TYPE csp_case_closing_rfid_status_enum :
(
	CSP_CASE_CLOSING_RFID_STATUS_START									:= 5,
	CSP_CASE_CLOSING_RFID_STATUS_ENABLED								:= 6,
	CSP_CASE_CLOSING_RFID_STATUS_PADDLES_START							:= 10,
	CSP_CASE_CLOSING_RFID_STATUS_VERIFY_AXIS_SAFE_POS					:= 15,
	CSP_CASE_CLOSING_RFID_STATUS_UPPER_START 							:= 20,
	CSP_CASE_CLOSING_RFID_STATUS_UPPER_VERIFY_AXIS_POS					:= 25,
	CSP_CASE_CLOSING_RFID_STATUS_UPPER_READ_START						:= 30,
	CSP_CASE_CLOSING_RFID_STATUS_UPPER_READ_CHECK_RESULT				:= 35,
	CSP_CASE_CLOSING_RFID_STATUS_UPPER_RETURN_TO_SAFE_POS				:= 40,
	CSP_CASE_CLOSING_RFID_STATUS_UPPER_READ_DONE						:= 45,
	
	CSP_CASE_CLOSING_RFID_STATUS_LOWER_START 							:= 50,
	CSP_CASE_CLOSING_RFID_STATUS_LOWER_VERIFY_AXIS_POS					:= 55,
	CSP_CASE_CLOSING_RFID_STATUS_LOWER_READ_START						:= 60,
	CSP_CASE_CLOSING_RFID_STATUS_LOWER_READ_CHECK_RESULT				:= 65,
	CSP_CASE_CLOSING_RFID_STATUS_LOWER_RETURN_TO_SAFE_POS				:= 70,
	CSP_CASE_CLOSING_RFID_STATUS_LOWER_READ_DONE						:= 75,
	
	
	CSP_CASE_CLOSING_RFID_STATUS_VERIFY_VALUES							:= 100,
		
	CSP_CASE_CLOSING_RFID_STATUS_COMPLETE								:= 220,
	
	CSP_CASE_CLOSING_RFID_STATUS_ERROR									:= 666,
			
	CSP_CASE_CLOSING_RFID_STATUS_WAITING								:= 900
	
) := CSP_CASE_CLOSING_RFID_STATUS_START;
END_TYPE

(* stored: Version 1.1.0.1, ProductVersion 3.1.4024.3
   DUT csp_case_closing_rfid_status_enum: Id {4f172b95-9a9e-0462-0b71-1e1d70df77b7} *)
